PROGRAM MAIN
VAR
	sanityCheck : int;
END_VAR

sanityCheck:=sanityCheck+1;

END_PROGRAM

(* stored: Version 1.1.0.1, ProductVersion 3.1.4024.15
   POU MAIN: Id {66d4f454-7bbd-49ec-95c5-88132eb8edd7}, SpecialFunc None *)
